(* Logix 5000 project; controller Safety vendor 1 type 14 code 148 rev 32.11; software revision 32.03; part 10 of 17 *)
(* tags used below, declared in another part *)
   ChgMe : BOOL;
   EnBridle_DrvsOff : BOOL;   // Entry Bridle Drives OFF ( 1= OFF)
   EnBridle_SafeOffEn : BOOL;   // Entry Bridle Safe-Off Enable ( 1= Enable )
   EnBridle_SafeOffFltRst : BOOL;   // Entry Bridle Safe-Off Fault Reset ( 1= Reset Cmd )
   ESTOP_x311PB130 : DCI_STOP;   // OS14 Shear Estop Pushbutton
   ESTOP_x311PB130_Flt : ALIAS FOR Flt_Estops.17;   // OS14 Shear EStop Pushbutton Fault ( 1= Fault)
   Flt_Modules : DINT[5];   // Point IO Module Fault Word
   FltsToCitect : DINT[64];   // Faults to Citect
   Line_TotalMode : BOOL;   // Line TOTAL Mode ( 1= Total Mode) (0 = Coil to Coil)
   LineSts : UDT_SysStatus;
   MCC1_S1_ModFlt : ALIAS FOR Flt_Modules[2].0;   // MCC1 Point I/O Slot01 Module Fault (1 = Fault)
   MCC1_S6_ModFlt : ALIAS FOR Flt_Modules[2].1;   // MCC1 Point I/O Slot06 Module Fault (1 = Fault)
   MCC2_S1_ModFlt : ALIAS FOR Flt_Modules[2].2;   // MCC2 Point I/O Slot01 Module Fault (1 = Fault)
   MCC2_S2_ModFlt : ALIAS FOR Flt_Modules[2].3;   // MCC2 Point I/O Slot02 Module Fault (1 = Fault)
   MCC3_S1_ModFlt : ALIAS FOR Flt_Modules[2].4;   // MCC3 Point I/O Slot01 Module Fault (1 = Fault)
   MCC3_S3_ModFlt : ALIAS FOR Flt_Modules[2].5;   // MCC3 Point I/O Slot03 Module Fault (1 = Fault)
   MCC3_S4_ModFlt : ALIAS FOR Flt_Modules[2].6;   // MCC3 Point I/O Slot04 Module Fault (1 = Fault)
   MCC4_S1_ModFlt : ALIAS FOR Flt_Modules[2].7;   // MCC4 Point I/O Slot01 Module Fault (1 = Fault)
   MCC4_S3_ModFlt : ALIAS FOR Flt_Modules[2].8;   // MCC4 Point I/O Slot03 Module Fault (1 = Fault)
   MCC4_S4_ModFlt : ALIAS FOR Flt_Modules[2].9;   // MCC4 Point I/O Slot04 Module Fault (1 = Fault)
   MCC5_S1_ModFlt : ALIAS FOR Flt_Modules[2].10;   // MCC5 Point I/O Slot01 Module Fault (1 = Fault)
   MCC5_S3_ModFlt : ALIAS FOR Flt_Modules[2].11;   // MCC5 Point I/O Slot03 Module Fault (1 = Fault)
   MCC5_S4_ModFlt : ALIAS FOR Flt_Modules[2].12;   // MCC5 Point I/O Slot04 Module Fault (1 = Fault)
   MCC5_S5_ModFlt : ALIAS FOR Flt_Modules[2].13;   // MCC5 Point I/O Slot05 Module Fault (1 = Fault)
   OS14_FltRstCmd : BOOL;   // OS14 Fault Reset Command ( 1= Reset Cmd)
   OS14_Shear_EstopRstCmd : BOOL;   // OS14_Shear Estop Reset Command ( 1= Reset Cmd)
   OS14_Shear_FltRstCmd : BOOL;   // OS14_Shear Fault Reset Command ( 1= Reset Cmd)
   OS14_Shear_No_EStops : BOOL;   // OS14_Shear No Estops ( 1= OK)
   PrCon_DrvsOff : BOOL;   // Product Conveyors (1-3) Drives OFF ( 1= OFF)
   PW_DrvsOff : BOOL;   // Paper Winder Drives OFF ( 1= OFF)
   SafeOff_y172CR460 : CONFIGURABLE_ROUT;   // Shear Die Main Contactor Relay
   SafeOff_y613CR460 : CONFIGURABLE_ROUT;   // Unwind Op Side Main Contactor Relay
   SafeOff_y613CR460_Flt : ALIAS FOR Flt_SafeOff[0].2;   // Unwind Op Side Main Contactor Relay Fault ( 1= Fault)
   SafeOff_y613CR510 : CONFIGURABLE_ROUT;   // Unwind Op Side Drive Enable Relay
   SafeOff_y613CR510_Flt : ALIAS FOR Flt_SafeOff[0].3;   // Unwind Op Side Drive Enable Relay Fault ( 1= Fault)
   SafeOff_y613CR550 : CONFIGURABLE_ROUT;   // Unwind Drive Side Main Contactor Relay
   SafeOff_y613CR550_Flt : ALIAS FOR Flt_SafeOff[0].4;   // Unwind Drive Side Main Contactor Relay Fault ( 1= Fault)
   SafeOff_y613CR590 : CONFIGURABLE_ROUT;   // Unwind Drive Side Drive Enable Relay
   SafeOff_y613CR590_Flt : ALIAS FOR Flt_SafeOff[0].5;   // Unwind Drive Side Drive Enable Relay Fault ( 1= Fault)
   SafeOff_y613CR630 : CONFIGURABLE_ROUT;   // #1 Entry Bridle Roll 2 Main Contactor Relay
   SafeOff_y613CR630_Flt : ALIAS FOR Flt_SafeOff[0].6;   // #1 Entry Bridle Roll 2 Main Contactor Relay Fault ( 1= Fault)
   SafeOff_y613CR670 : CONFIGURABLE_ROUT;   // #1 Entry Bridle Roll 2 Drive Enable Relay
   SafeOff_y613CR670_Flt : ALIAS FOR Flt_SafeOff[0].7;   // #1 Entry Bridle Roll 2 Drive Enable Relay Fault ( 1= Fault)
   SafeOff_y613CR710 : CONFIGURABLE_ROUT;   // #2 Entry Bridle Roll 3 Main Contactor Relay
   SafeOff_y613CR710_Flt : ALIAS FOR Flt_SafeOff[0].8;   // #2 Entry Bridle Roll 3 Main Contactor Relay Fault ( 1= Fault)
   SafeOff_y613CR750 : CONFIGURABLE_ROUT;   // #2 Entry Bridle Roll 3 Drive Enable Relay
   SafeOff_y613CR750_Flt : ALIAS FOR Flt_SafeOff[0].9;   // #2 Entry Bridle Roll 3 Drive Enable Relay Fault ( 1= Fault)
   SafeOff_y614CR040 : CONFIGURABLE_ROUT;   // #1 Exit Bridle Roll 6 Main Contactor Relay
   SafeOff_y614CR210 : CONFIGURABLE_ROUT;   // Rewind Main Contactor Relay
   SC_DrvsOff : BOOL;   // Scrap Chop Conveyor Drives OFF ( 1= OFF)
   ScInCon_DrvsOff : BOOL;   // Scrap Incline Conveyor Drives OFF ( 1= OFF)
   SGWA_DrvsOff : BOOL;   // Side Guide Width Adjust Drives OFF ( 1= OFF)
   ShearSts : UDT_ShearStatus;
   SkBkSt_DrvsOff : BOOL;   // Stacker Backstop Drives OFF ( 1= OFF)
   SkBlwr_DrvsOff : BOOL;   // Stacker Blower Drives OFF ( 1= OFF)
   Sr_DrvsOff : BOOL;   // Shear Pinch Roll/ Metering Back Up Drives OFF ( 1= OFF)
   SrCon_DrvsOff : BOOL;   // Shear Conveyor Drives OFF ( 1= OFF)
   StPR_DrvsOff : BOOL;   // Sheeter Pinch Roll Drives OFF ( 1= OFF)
   TK_DrvsOff : BOOL;   // Trimmer Knives/ Width Adjust Drives OFF ( 1= OFF)
   UnPR_DrvsOff : BOOL;   // Unwind Pinch Roll Drives OFF ( 1= OFF)
   UNW_DrvsOff : BOOL;   // Unwind Drives OFF ( 1= OFF)
   UNW_SafeOffEn : BOOL;   // Unwind Safe-Off Enable ( 1= Enable )
   UNW_SafeOffFltRst : BOOL;   // Unwind Safe-Off Fault Reset ( 1= Reset Cmd )
   WTPR_DrvsOff : BOOL;   // Wash Tank Pinch Rolls (1-4) Drives OFF ( 1= OFF)
   x311PB130a : ALIAS FOR OS14:1:I.Pt02Data;   // Shear Emergency Stop PB Os14
   x311PB130b : ALIAS FOR OS14:1:I.Pt03Data;   // Shear Emergency Stop PB Os14
   x613CR460 : ALIAS FOR CHPLC:1:I.Pt00Data;   // Unwind Operator Side Main Contactor Safety Relay
   x613CR510 : ALIAS FOR CHPLC:1:I.Pt01Data;   // Unwind Operator Side Drive Enable Safety Relay
   x613CR550 : ALIAS FOR CHPLC:1:I.Pt02Data;   // Unwind Drive Side Main Contactor Safety Relay
   x613CR590 : ALIAS FOR CHPLC:1:I.Pt03Data;   // Unwind Drive Side Drive Enable Safety Relay
   x613CR630 : ALIAS FOR CHPLC:1:I.Pt04Data;   // #1 Entry Bridle Roll 2 Main Contactor Safety Relay
   x613CR670 : ALIAS FOR CHPLC:1:I.Pt05Data;   // #1 Entry Bridle Roll 2 Drive Enable Safety Relay
   x613CR710 : ALIAS FOR CHPLC:1:I.Pt06Data;   // #2 Entry Bridle Roll 3 Main Contactor Safety Relay
   x613CR750 : ALIAS FOR CHPLC:1:I.Pt07Data;   // #2 Entry Bridle Roll 3 Drive Enable Safety Relay
   y613CR460 : ALIAS FOR CHPLC:4:O.Pt00Data;   // Unwind Operator Side Main Contactor Safety Relay
   y613CR510 : ALIAS FOR CHPLC:4:O.Pt01Data;   // Unwind Operator Side Drive Enable Safety Relay
   y613CR550 : ALIAS FOR CHPLC:4:O.Pt02Data;   // Unwind Drive Side Main Contactor Safety Relay
   y613CR590 : ALIAS FOR CHPLC:4:O.Pt03Data;   // Unwind Drive Side Drive Enable Safety Relay
   y613CR630 : ALIAS FOR CHPLC:4:O.Pt04Data;   // #1 Entry Bridle Roll 2 Main Contactor Safety Relay
   y613CR670 : ALIAS FOR CHPLC:4:O.Pt05Data;   // #1 Entry Bridle Roll 2 Drive Enable Safety Relay
   y613CR710 : ALIAS FOR CHPLC:4:O.Pt06Data;   // #2 Entry Bridle Roll 3 Main Contactor Safety Relay
   y613CR750 : ALIAS FOR CHPLC:4:O.Pt07Data;   // #2 Entry Bridle Roll 3 Drive Enable Safety Relay
(* Estops, continued *)

ROUTINE C00_OS14_Shear_EStop   (* ladder *)
// OS14 Shear EStop
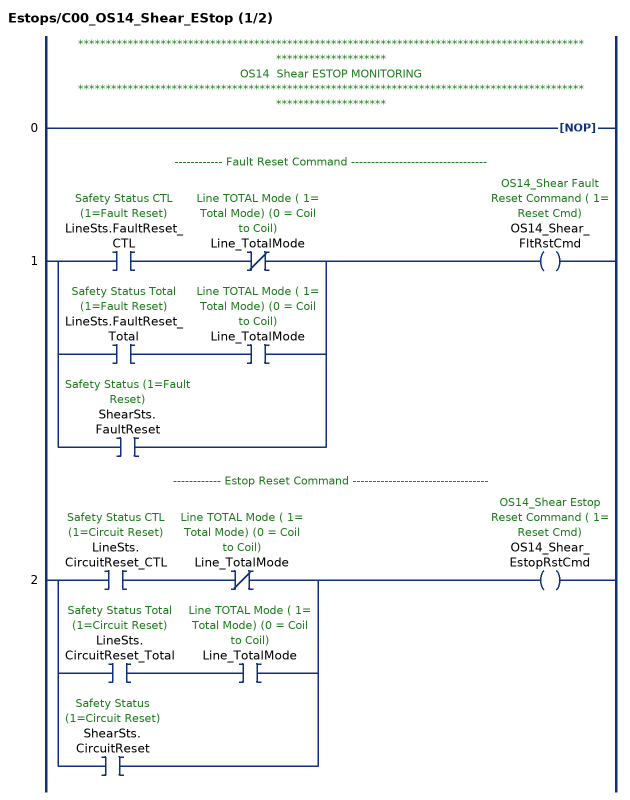
   // ****************************************************************************************************************
   // OS14  Shear ESTOP MONITORING
   // ****************************************************************************************************************
   0: NOP();
   // ------------ Fault Reset Command ----------------------------------
   1: [XIC(LineSts.FaultReset_CTL) XIO(Line_TotalMode) ,XIC(LineSts.FaultReset_Total) XIC(Line_TotalMode) ,XIC(ShearSts.FaultReset) ]OTE(OS14_Shear_FltRstCmd);
   // ------------ Estop Reset Command ----------------------------------
   2: [XIC(LineSts.CircuitReset_CTL) XIO(Line_TotalMode) ,XIC(LineSts.CircuitReset_Total) XIC(Line_TotalMode) ,XIC(ShearSts.CircuitReset) ]OTE(OS14_Shear_EstopRstCmd);
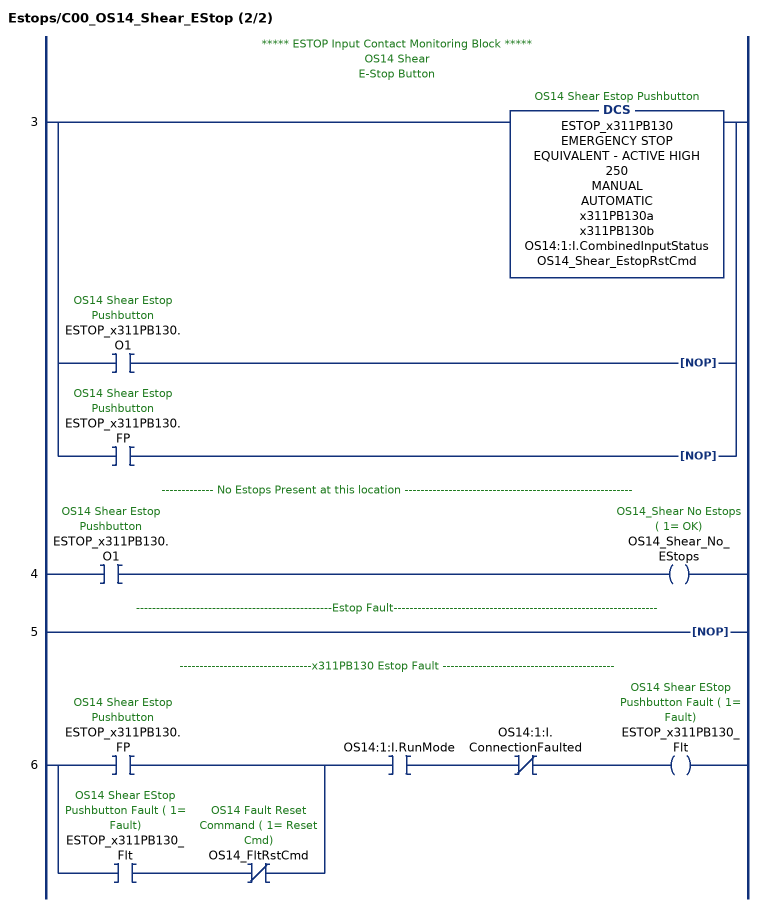
   // ***** ESTOP Input Contact Monitoring Block *****
   // OS14 Shear
   // E-Stop Button
   3: [DCS(ESTOP_x311PB130,EMERGENCY STOP,EQUIVALENT - ACTIVE HIGH,250,MANUAL,AUTOMATIC,x311PB130a,x311PB130b,OS14:1:I.CombinedInputStatus,OS14_Shear_EstopRstCmd) ,XIC(ESTOP_x311PB130.O1) NOP() ,XIC(ESTOP_x311PB130.FP) NOP() ];
   // ------------- No Estops Present at this location ---------------------------------------------------------
   4: XIC(ESTOP_x311PB130.O1)OTE(OS14_Shear_No_EStops);
   // -------------------------------------------------Estop Fault------------------------------------------------------------------
   5: NOP();
   // ---------------------------------x311PB130 Estop Fault -------------------------------------------
   6: [XIC(ESTOP_x311PB130.FP) ,XIC(ESTOP_x311PB130_Flt) XIO(OS14_FltRstCmd) ]XIC(OS14:1:I.RunMode)XIO(OS14:1:I.ConnectionFaulted)OTE(ESTOP_x311PB130_Flt);
END_ROUTINE
END_PROGRAM

PROGRAM JUNK   (* main routine SCRATCH *)

ROUTINE JUNKY   (* ladder *)
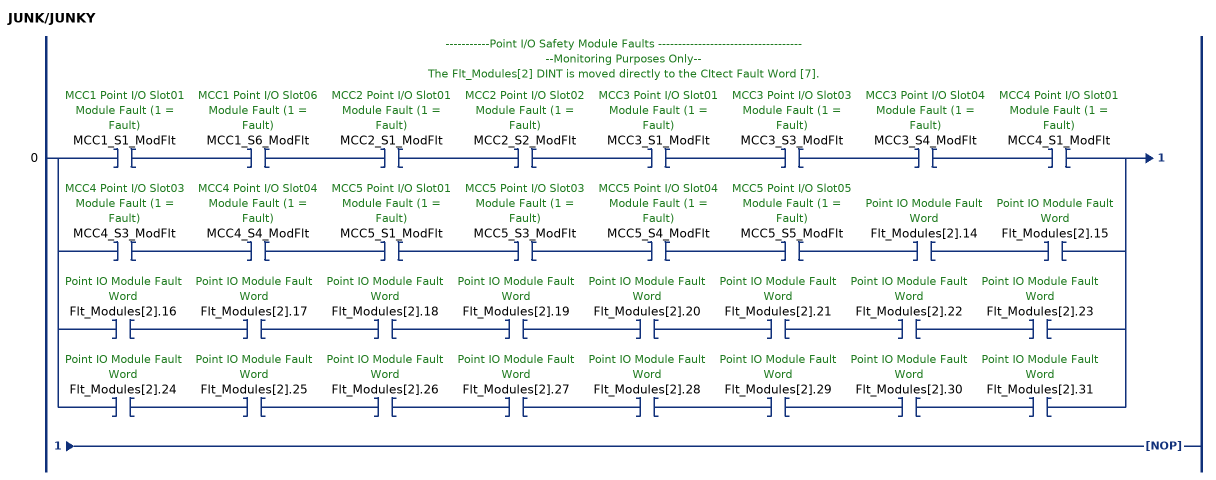
   // -----------Point I/O Safety Module Faults ------------------------------------
   // --Monitoring Purposes Only--
   // The Flt_Modules[2] DINT is moved directly to the CItect Fault Word [7].
   0: [XIC(MCC1_S1_ModFlt) XIC(MCC1_S6_ModFlt) XIC(MCC2_S1_ModFlt) XIC(MCC2_S2_ModFlt) XIC(MCC3_S1_ModFlt) XIC(MCC3_S3_ModFlt) XIC(MCC3_S4_ModFlt) XIC(MCC4_S1_ModFlt) ,XIC(MCC4_S3_ModFlt) XIC(MCC4_S4_ModFlt) XIC(MCC5_S1_ModFlt) XIC(MCC5_S3_ModFlt) XIC(MCC5_S4_ModFlt) XIC(MCC5_S5_ModFlt) XIC(Flt_Modules[2].14) XIC(Flt_Modules[2].15) ,XIC(Flt_Modules[2].16) XIC(Flt_Modules[2].17) XIC(Flt_Modules[2].18) XIC(Flt_Modules[2].19) XIC(Flt_Modules[2].20) XIC(Flt_Modules[2].21) XIC(Flt_Modules[2].22) XIC(Flt_Modules[2].23) ,XIC(Flt_Modules[2].24) XIC(Flt_Modules[2].25) XIC(Flt_Modules[2].26) XIC(Flt_Modules[2].27) XIC(Flt_Modules[2].28) XIC(Flt_Modules[2].29) XIC(Flt_Modules[2].30) XIC(Flt_Modules[2].31) ]NOP();
END_ROUTINE

ROUTINE SCRATCH   (* ladder *)
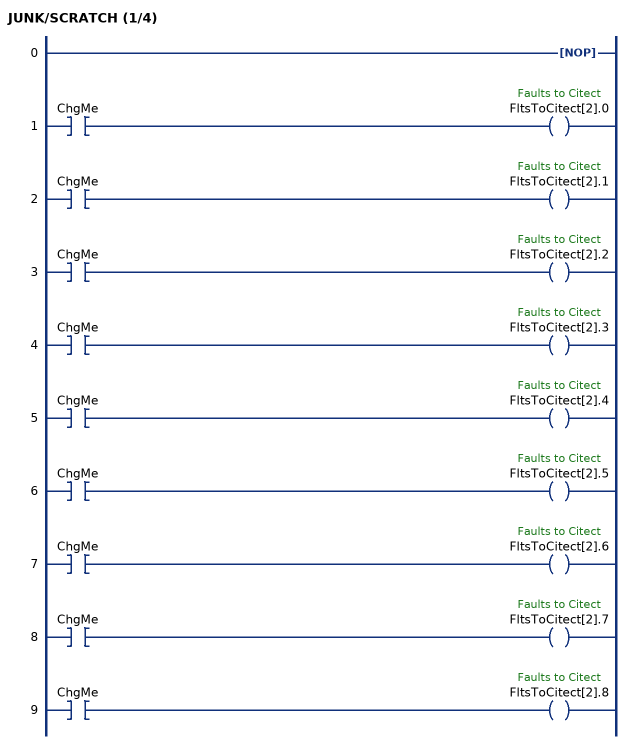
   0: NOP();
   1: XIC(ChgMe)OTE(FltsToCitect[2].0);
   2: XIC(ChgMe)OTE(FltsToCitect[2].1);
   3: XIC(ChgMe)OTE(FltsToCitect[2].2);
   4: XIC(ChgMe)OTE(FltsToCitect[2].3);
   5: XIC(ChgMe)OTE(FltsToCitect[2].4);
   6: XIC(ChgMe)OTE(FltsToCitect[2].5);
   7: XIC(ChgMe)OTE(FltsToCitect[2].6);
   8: XIC(ChgMe)OTE(FltsToCitect[2].7);
   9: XIC(ChgMe)OTE(FltsToCitect[2].8);
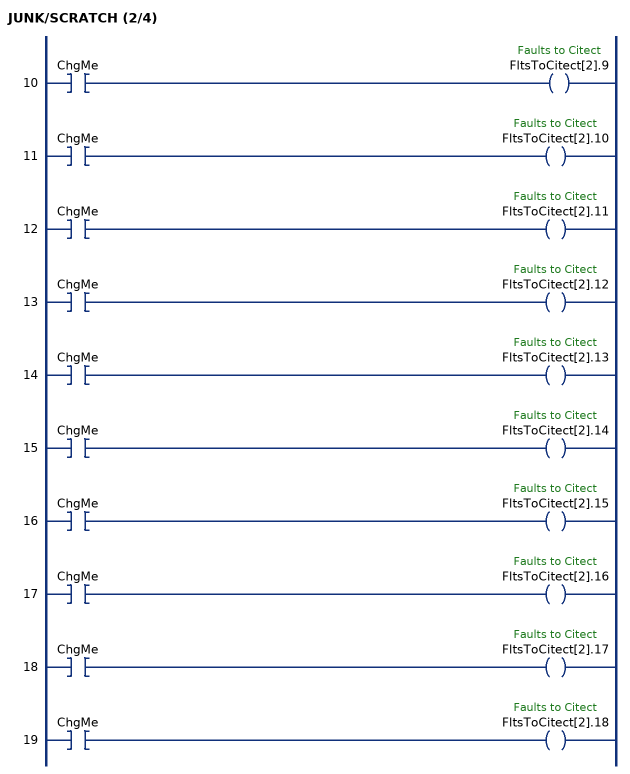
   10: XIC(ChgMe)OTE(FltsToCitect[2].9);
   11: XIC(ChgMe)OTE(FltsToCitect[2].10);
   12: XIC(ChgMe)OTE(FltsToCitect[2].11);
   13: XIC(ChgMe)OTE(FltsToCitect[2].12);
   14: XIC(ChgMe)OTE(FltsToCitect[2].13);
   15: XIC(ChgMe)OTE(FltsToCitect[2].14);
   16: XIC(ChgMe)OTE(FltsToCitect[2].15);
   17: XIC(ChgMe)OTE(FltsToCitect[2].16);
   18: XIC(ChgMe)OTE(FltsToCitect[2].17);
   19: XIC(ChgMe)OTE(FltsToCitect[2].18);
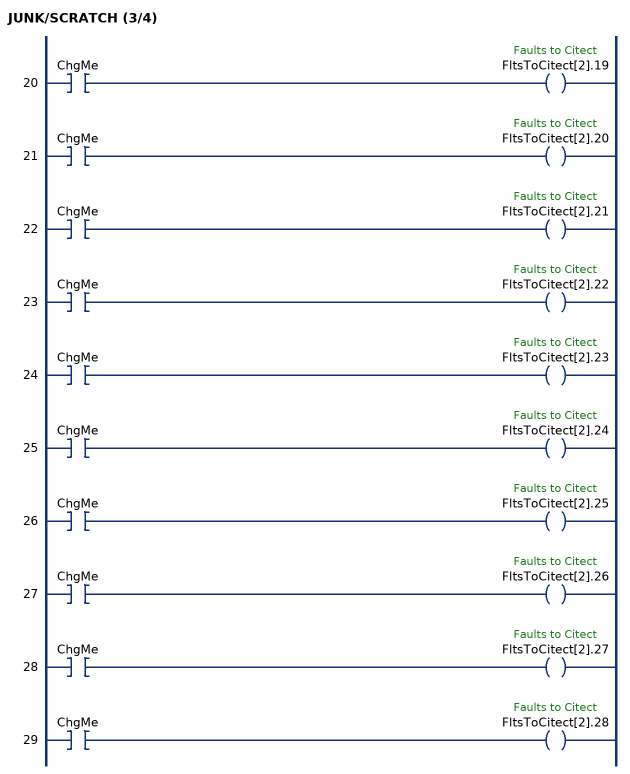
   20: XIC(ChgMe)OTE(FltsToCitect[2].19);
   21: XIC(ChgMe)OTE(FltsToCitect[2].20);
   22: XIC(ChgMe)OTE(FltsToCitect[2].21);
   23: XIC(ChgMe)OTE(FltsToCitect[2].22);
   24: XIC(ChgMe)OTE(FltsToCitect[2].23);
   25: XIC(ChgMe)OTE(FltsToCitect[2].24);
   26: XIC(ChgMe)OTE(FltsToCitect[2].25);
   27: XIC(ChgMe)OTE(FltsToCitect[2].26);
   28: XIC(ChgMe)OTE(FltsToCitect[2].27);
   29: XIC(ChgMe)OTE(FltsToCitect[2].28);
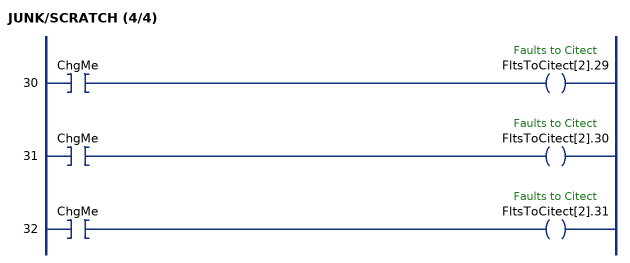
   30: XIC(ChgMe)OTE(FltsToCitect[2].29);
   31: XIC(ChgMe)OTE(FltsToCitect[2].30);
   32: XIC(ChgMe)OTE(FltsToCitect[2].31);
END_ROUTINE
END_PROGRAM

PROGRAM SafeOff   (* main routine A00_Main, safety *)

ROUTINE A00_Main   (* ladder *)
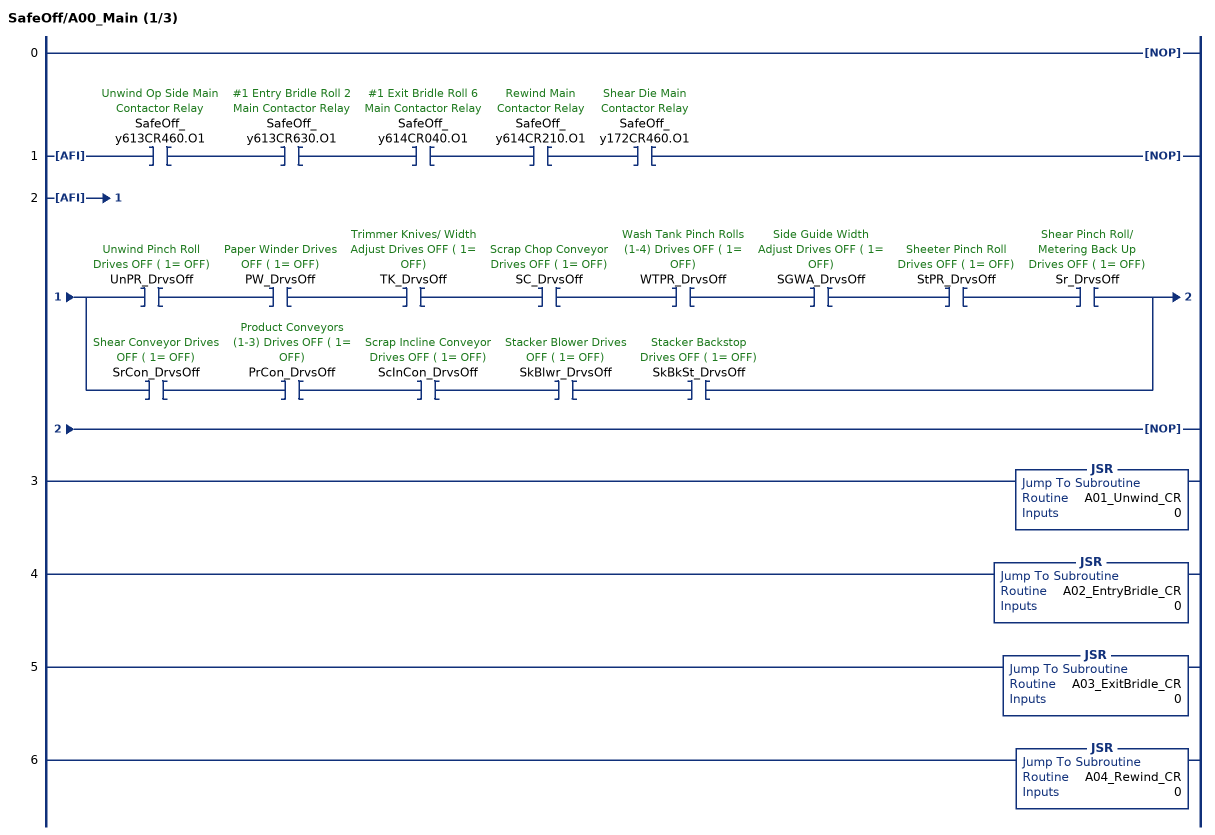
   0: NOP();
   1: AFI()XIC(SafeOff_y613CR460.O1)XIC(SafeOff_y613CR630.O1)XIC(SafeOff_y614CR040.O1)XIC(SafeOff_y614CR210.O1)XIC(SafeOff_y172CR460.O1)NOP();
   2: AFI()[XIC(UnPR_DrvsOff) XIC(PW_DrvsOff) XIC(TK_DrvsOff) XIC(SC_DrvsOff) XIC(WTPR_DrvsOff) XIC(SGWA_DrvsOff) XIC(StPR_DrvsOff) XIC(Sr_DrvsOff) ,XIC(SrCon_DrvsOff) XIC(PrCon_DrvsOff) XIC(ScInCon_DrvsOff) XIC(SkBlwr_DrvsOff) XIC(SkBkSt_DrvsOff) ]NOP();
   3: JSR(A01_Unwind_CR,0);
   4: JSR(A02_EntryBridle_CR,0);
   5: JSR(A03_ExitBridle_CR,0);
   6: JSR(A04_Rewind_CR,0);
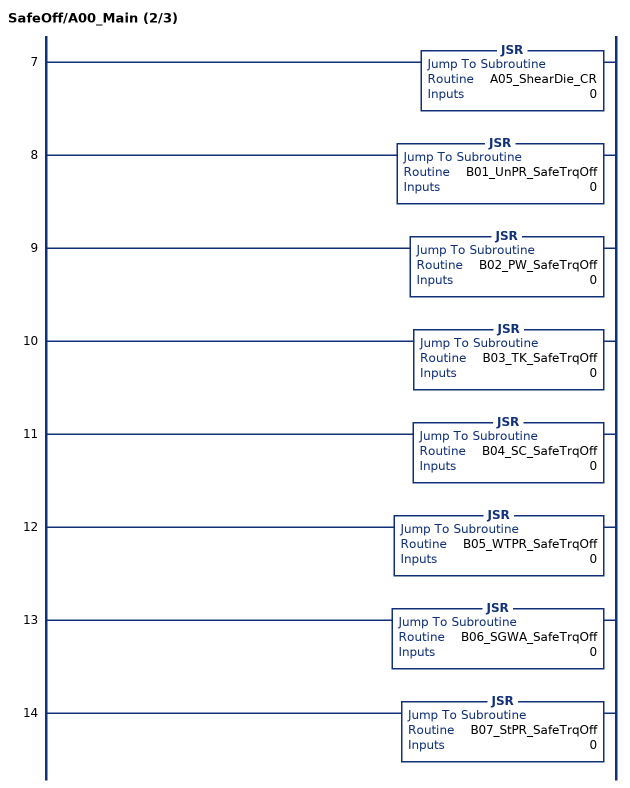
   7: JSR(A05_ShearDie_CR,0);
   8: JSR(B01_UnPR_SafeTrqOff,0);
   9: JSR(B02_PW_SafeTrqOff,0);
   10: JSR(B03_TK_SafeTrqOff,0);
   11: JSR(B04_SC_SafeTrqOff,0);
   12: JSR(B05_WTPR_SafeTrqOff,0);
   13: JSR(B06_SGWA_SafeTrqOff,0);
   14: JSR(B07_StPR_SafeTrqOff,0);
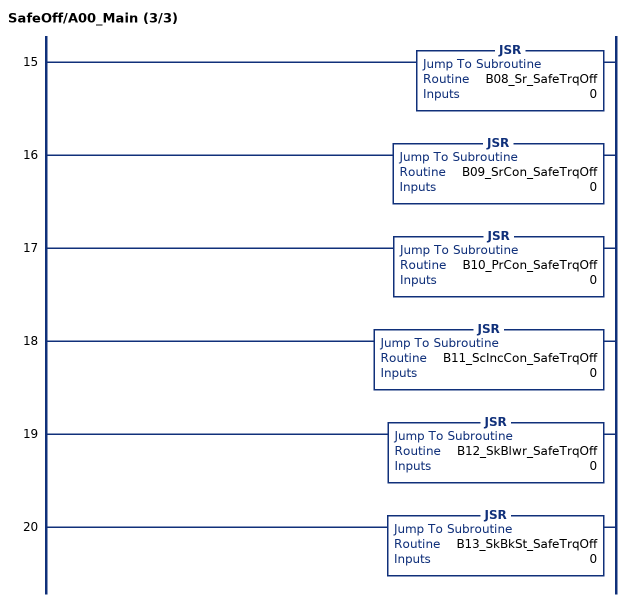
   15: JSR(B08_Sr_SafeTrqOff,0);
   16: JSR(B09_SrCon_SafeTrqOff,0);
   17: JSR(B10_PrCon_SafeTrqOff,0);
   18: JSR(B11_ScIncCon_SafeTrqOff,0);
   19: JSR(B12_SkBlwr_SafeTrqOff,0);
   20: JSR(B13_SkBkSt_SafeTrqOff,0);
END_ROUTINE

ROUTINE A01_Unwind_CR   (* ladder *)
// Unwind
// Main Contactor and Drive Enable
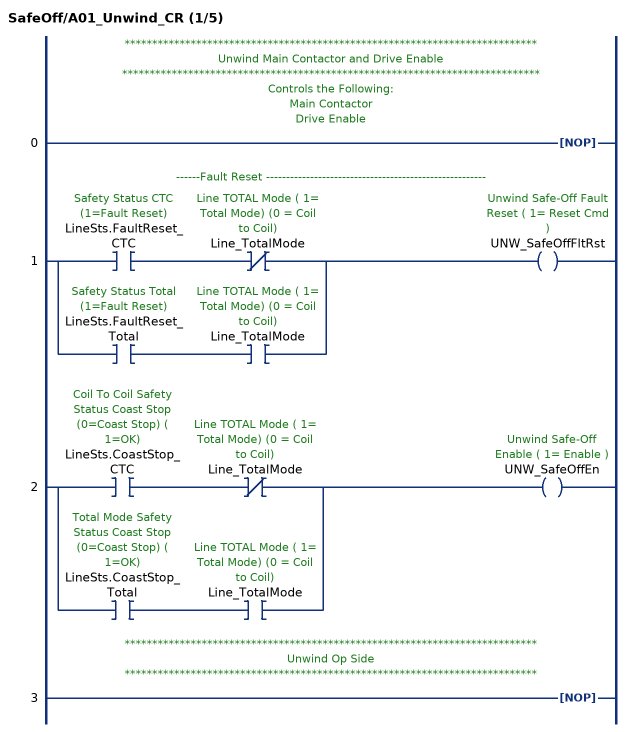
   // ***************************************************************************
   // Unwind Main Contactor and Drive Enable
   // ****************************************************************************
   // Controls the Following:
   // Main Contactor
   // Drive Enable
   0: NOP();
   // ------Fault Reset -------------------------------------------------------
   1: [XIC(LineSts.FaultReset_CTC) XIO(Line_TotalMode) ,XIC(LineSts.FaultReset_Total) XIC(Line_TotalMode) ]OTE(UNW_SafeOffFltRst);
   2: [XIC(LineSts.CoastStop_CTC) XIO(Line_TotalMode) ,XIC(LineSts.CoastStop_Total) XIC(Line_TotalMode) ]OTE(UNW_SafeOffEn);
   // ***************************************************************************
   // Unwind Op Side
   // ***************************************************************************
   3: NOP();
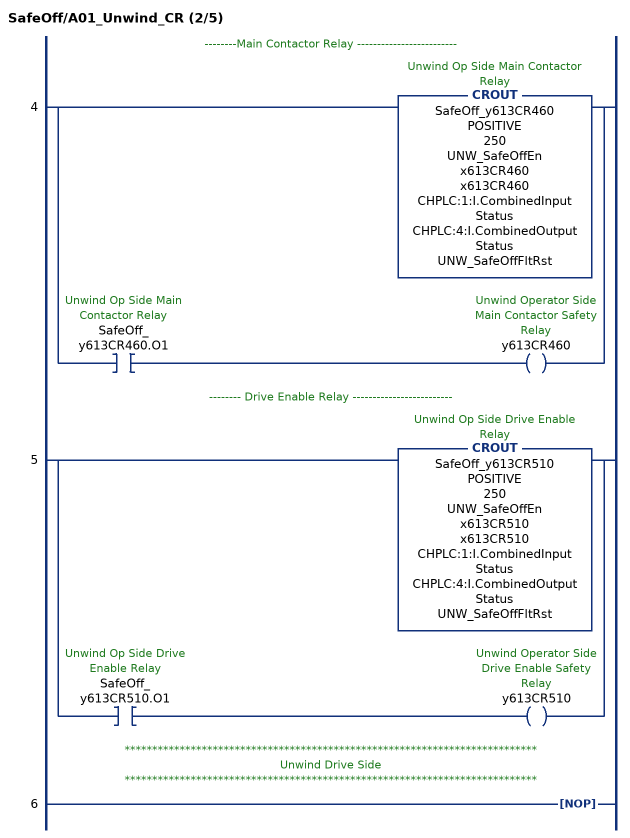
   // --------Main Contactor Relay -------------------------
   4: [CROUT(SafeOff_y613CR460,POSITIVE,250,UNW_SafeOffEn,x613CR460,x613CR460,CHPLC:1:I.CombinedInputStatus,CHPLC:4:I.CombinedOutputStatus,UNW_SafeOffFltRst) ,XIC(SafeOff_y613CR460.O1) OTE(y613CR460) ];
   // -------- Drive Enable Relay -------------------------
   5: [CROUT(SafeOff_y613CR510,POSITIVE,250,UNW_SafeOffEn,x613CR510,x613CR510,CHPLC:1:I.CombinedInputStatus,CHPLC:4:I.CombinedOutputStatus,UNW_SafeOffFltRst) ,XIC(SafeOff_y613CR510.O1) OTE(y613CR510) ];
   // ***************************************************************************
   // Unwind Drive Side
   // ***************************************************************************
   6: NOP();
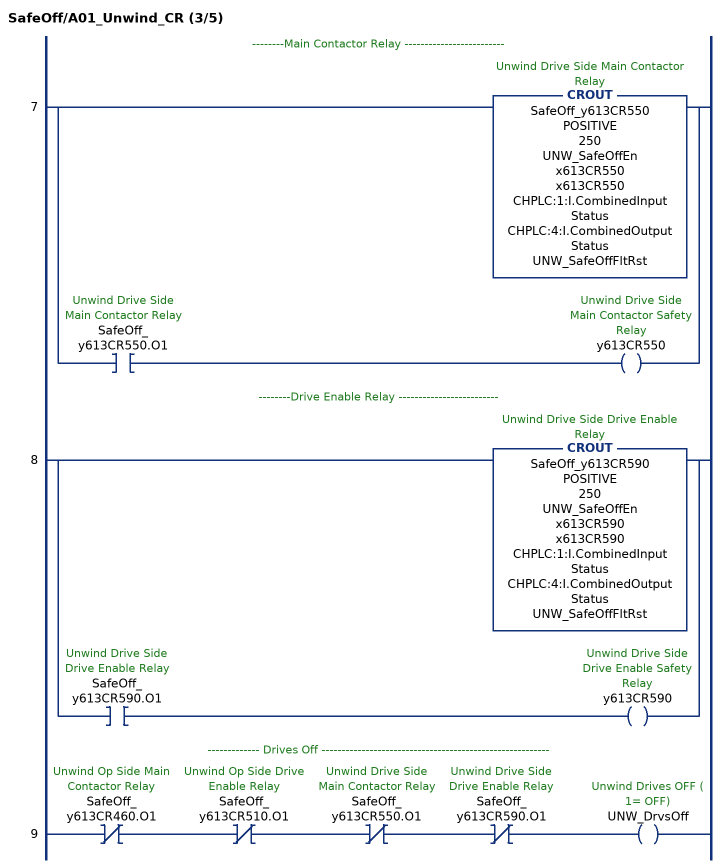
   // --------Main Contactor Relay -------------------------
   7: [CROUT(SafeOff_y613CR550,POSITIVE,250,UNW_SafeOffEn,x613CR550,x613CR550,CHPLC:1:I.CombinedInputStatus,CHPLC:4:I.CombinedOutputStatus,UNW_SafeOffFltRst) ,XIC(SafeOff_y613CR550.O1) OTE(y613CR550) ];
   // --------Drive Enable Relay -------------------------
   8: [CROUT(SafeOff_y613CR590,POSITIVE,250,UNW_SafeOffEn,x613CR590,x613CR590,CHPLC:1:I.CombinedInputStatus,CHPLC:4:I.CombinedOutputStatus,UNW_SafeOffFltRst) ,XIC(SafeOff_y613CR590.O1) OTE(y613CR590) ];
   // ------------- Drives Off ---------------------------------------------------------
   9: XIO(SafeOff_y613CR460.O1)XIO(SafeOff_y613CR510.O1)XIO(SafeOff_y613CR550.O1)XIO(SafeOff_y613CR590.O1)OTE(UNW_DrvsOff);
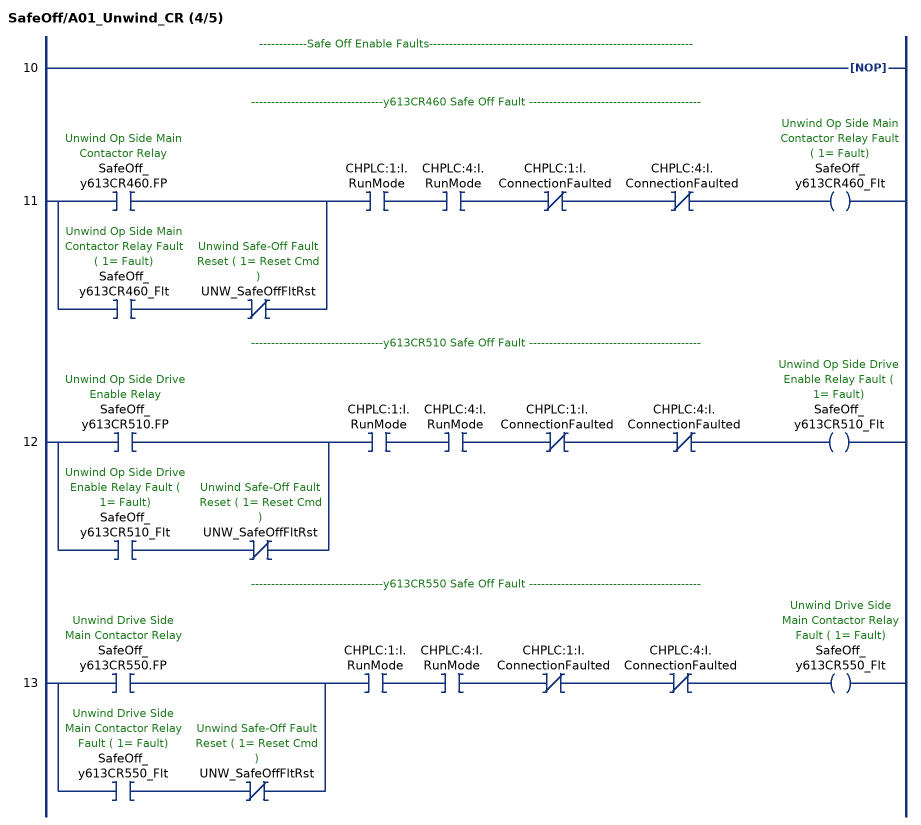
   // ------------Safe Off Enable Faults------------------------------------------------------------------
   10: NOP();
   // ---------------------------------y613CR460 Safe Off Fault -------------------------------------------
   11: [XIC(SafeOff_y613CR460.FP) ,XIC(SafeOff_y613CR460_Flt) XIO(UNW_SafeOffFltRst) ]XIC(CHPLC:1:I.RunMode)XIC(CHPLC:4:I.RunMode)XIO(CHPLC:1:I.ConnectionFaulted)XIO(CHPLC:4:I.ConnectionFaulted)OTE(SafeOff_y613CR460_Flt);
   // ---------------------------------y613CR510 Safe Off Fault -------------------------------------------
   12: [XIC(SafeOff_y613CR510.FP) ,XIC(SafeOff_y613CR510_Flt) XIO(UNW_SafeOffFltRst) ]XIC(CHPLC:1:I.RunMode)XIC(CHPLC:4:I.RunMode)XIO(CHPLC:1:I.ConnectionFaulted)XIO(CHPLC:4:I.ConnectionFaulted)OTE(SafeOff_y613CR510_Flt);
   // ---------------------------------y613CR550 Safe Off Fault -------------------------------------------
   13: [XIC(SafeOff_y613CR550.FP) ,XIC(SafeOff_y613CR550_Flt) XIO(UNW_SafeOffFltRst) ]XIC(CHPLC:1:I.RunMode)XIC(CHPLC:4:I.RunMode)XIO(CHPLC:1:I.ConnectionFaulted)XIO(CHPLC:4:I.ConnectionFaulted)OTE(SafeOff_y613CR550_Flt);
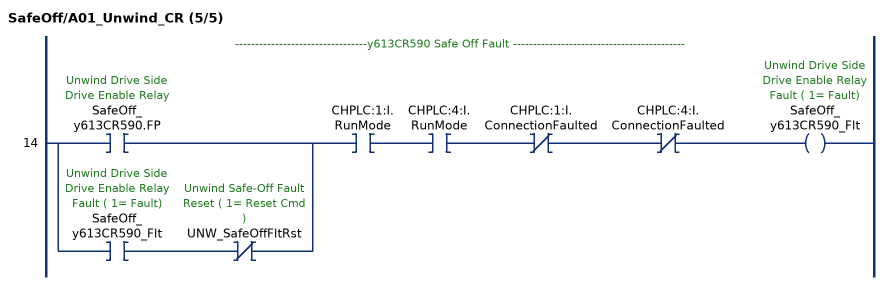
   // ---------------------------------y613CR590 Safe Off Fault -------------------------------------------
   14: [XIC(SafeOff_y613CR590.FP) ,XIC(SafeOff_y613CR590_Flt) XIO(UNW_SafeOffFltRst) ]XIC(CHPLC:1:I.RunMode)XIC(CHPLC:4:I.RunMode)XIO(CHPLC:1:I.ConnectionFaulted)XIO(CHPLC:4:I.ConnectionFaulted)OTE(SafeOff_y613CR590_Flt);
END_ROUTINE

ROUTINE A02_EntryBridle_CR   (* ladder *)
// Entry Bridle
// Main Contactor and Drive Enable
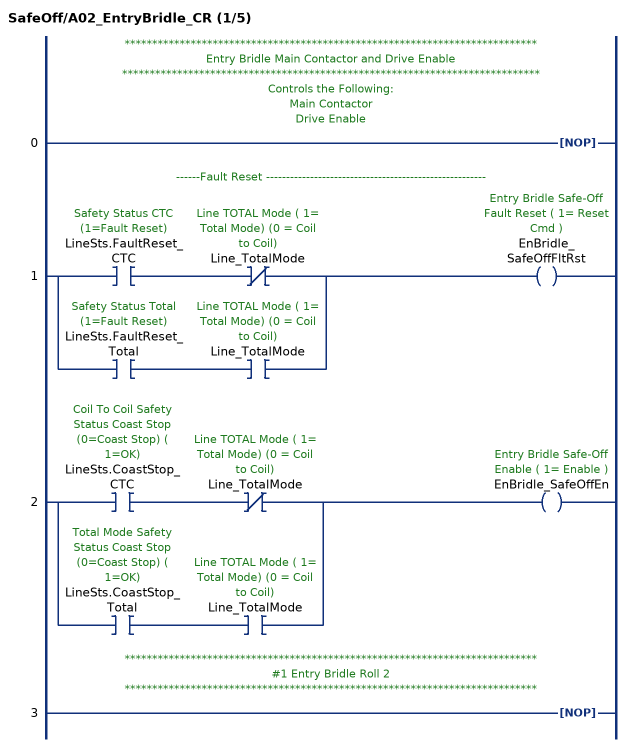
   // ***************************************************************************
   // Entry Bridle Main Contactor and Drive Enable
   // ****************************************************************************
   // Controls the Following:
   // Main Contactor
   // Drive Enable
   0: NOP();
   // ------Fault Reset -------------------------------------------------------
   1: [XIC(LineSts.FaultReset_CTC) XIO(Line_TotalMode) ,XIC(LineSts.FaultReset_Total) XIC(Line_TotalMode) ]OTE(EnBridle_SafeOffFltRst);
   2: [XIC(LineSts.CoastStop_CTC) XIO(Line_TotalMode) ,XIC(LineSts.CoastStop_Total) XIC(Line_TotalMode) ]OTE(EnBridle_SafeOffEn);
   // ***************************************************************************
   // #1 Entry Bridle Roll 2
   // ***************************************************************************
   3: NOP();
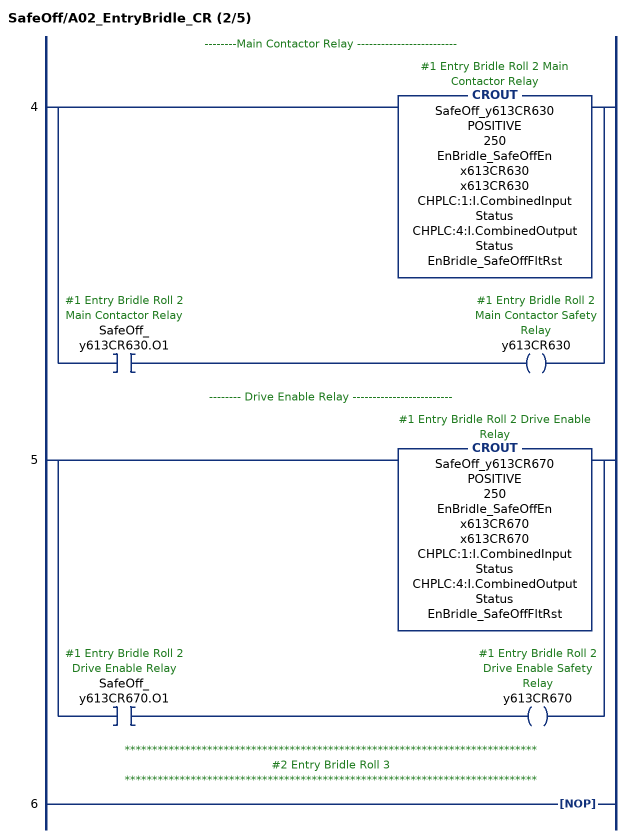
   // --------Main Contactor Relay -------------------------
   4: [CROUT(SafeOff_y613CR630,POSITIVE,250,EnBridle_SafeOffEn,x613CR630,x613CR630,CHPLC:1:I.CombinedInputStatus,CHPLC:4:I.CombinedOutputStatus,EnBridle_SafeOffFltRst) ,XIC(SafeOff_y613CR630.O1) OTE(y613CR630) ];
   // -------- Drive Enable Relay -------------------------
   5: [CROUT(SafeOff_y613CR670,POSITIVE,250,EnBridle_SafeOffEn,x613CR670,x613CR670,CHPLC:1:I.CombinedInputStatus,CHPLC:4:I.CombinedOutputStatus,EnBridle_SafeOffFltRst) ,XIC(SafeOff_y613CR670.O1) OTE(y613CR670) ];
   // ***************************************************************************
   // #2 Entry Bridle Roll 3
   // ***************************************************************************
   6: NOP();
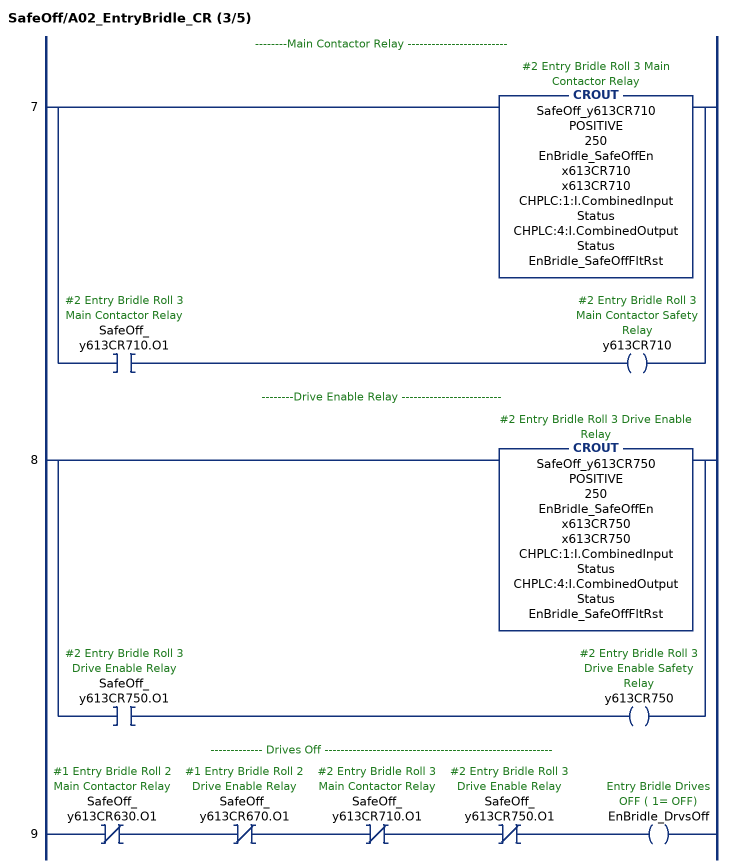
   // --------Main Contactor Relay -------------------------
   7: [CROUT(SafeOff_y613CR710,POSITIVE,250,EnBridle_SafeOffEn,x613CR710,x613CR710,CHPLC:1:I.CombinedInputStatus,CHPLC:4:I.CombinedOutputStatus,EnBridle_SafeOffFltRst) ,XIC(SafeOff_y613CR710.O1) OTE(y613CR710) ];
   // --------Drive Enable Relay -------------------------
   8: [CROUT(SafeOff_y613CR750,POSITIVE,250,EnBridle_SafeOffEn,x613CR750,x613CR750,CHPLC:1:I.CombinedInputStatus,CHPLC:4:I.CombinedOutputStatus,EnBridle_SafeOffFltRst) ,XIC(SafeOff_y613CR750.O1) OTE(y613CR750) ];
   // ------------- Drives Off ---------------------------------------------------------
   9: XIO(SafeOff_y613CR630.O1)XIO(SafeOff_y613CR670.O1)XIO(SafeOff_y613CR710.O1)XIO(SafeOff_y613CR750.O1)OTE(EnBridle_DrvsOff);
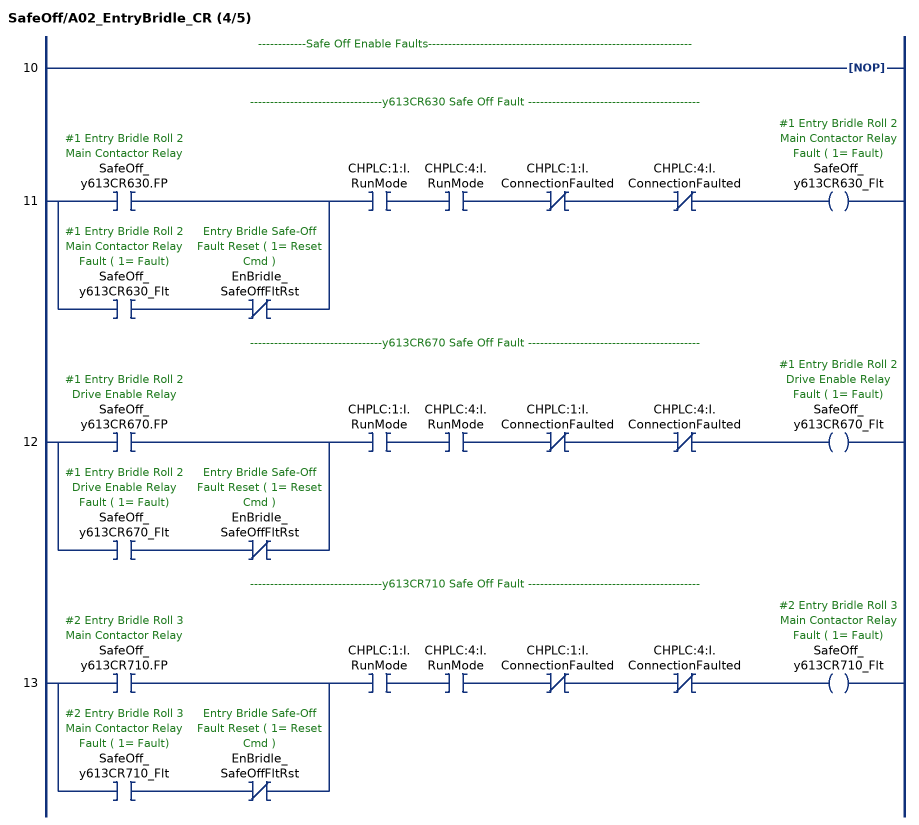
   // ------------Safe Off Enable Faults------------------------------------------------------------------
   10: NOP();
   // ---------------------------------y613CR630 Safe Off Fault -------------------------------------------
   11: [XIC(SafeOff_y613CR630.FP) ,XIC(SafeOff_y613CR630_Flt) XIO(EnBridle_SafeOffFltRst) ]XIC(CHPLC:1:I.RunMode)XIC(CHPLC:4:I.RunMode)XIO(CHPLC:1:I.ConnectionFaulted)XIO(CHPLC:4:I.ConnectionFaulted)OTE(SafeOff_y613CR630_Flt);
   // ---------------------------------y613CR670 Safe Off Fault -------------------------------------------
   12: [XIC(SafeOff_y613CR670.FP) ,XIC(SafeOff_y613CR670_Flt) XIO(EnBridle_SafeOffFltRst) ]XIC(CHPLC:1:I.RunMode)XIC(CHPLC:4:I.RunMode)XIO(CHPLC:1:I.ConnectionFaulted)XIO(CHPLC:4:I.ConnectionFaulted)OTE(SafeOff_y613CR670_Flt);
   // ---------------------------------y613CR710 Safe Off Fault -------------------------------------------
   13: [XIC(SafeOff_y613CR710.FP) ,XIC(SafeOff_y613CR710_Flt) XIO(EnBridle_SafeOffFltRst) ]XIC(CHPLC:1:I.RunMode)XIC(CHPLC:4:I.RunMode)XIO(CHPLC:1:I.ConnectionFaulted)XIO(CHPLC:4:I.ConnectionFaulted)OTE(SafeOff_y613CR710_Flt);
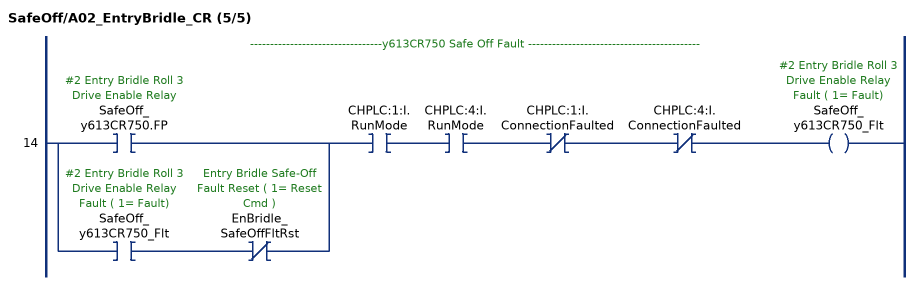
   // ---------------------------------y613CR750 Safe Off Fault -------------------------------------------
   14: [XIC(SafeOff_y613CR750.FP) ,XIC(SafeOff_y613CR750_Flt) XIO(EnBridle_SafeOffFltRst) ]XIC(CHPLC:1:I.RunMode)XIC(CHPLC:4:I.RunMode)XIO(CHPLC:1:I.ConnectionFaulted)XIO(CHPLC:4:I.ConnectionFaulted)OTE(SafeOff_y613CR750_Flt);
END_ROUTINE
